FUNCTION_BLOCK CSV_WRITER_4
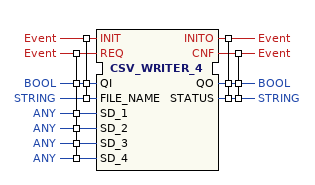
  EVENT_INPUT
    INIT WITH QI, FILE_NAME;
    REQ WITH QI, SD_1, SD_2, SD_3, SD_4;
  END_EVENT
  EVENT_OUTPUT
    INITO WITH QO, STATUS;
    CNF WITH QO, STATUS;
  END_EVENT
  VAR_INPUT
    QI : BOOL;
    FILE_NAME : STRING;
    SD_1 : ANY;
    SD_2 : ANY;
    SD_3 : ANY;
    SD_4 : ANY;
  END_VAR
  VAR_OUTPUT
    QO : BOOL;
    STATUS : STRING;
  END_VAR
END_FUNCTION_BLOCK
